FUNCTION_BLOCK FB_ActiveTarget EXTENDS FB_TargetBase IMPLEMENTS I_Device
VAR_INPUT
END_VAR
VAR_OUTPUT
END_VAR
VAR
	bInitFB			: BOOL := TRUE;
	nNotifyId		: UINT;
	bError			: BOOL;
	nErrorId		: ERRORID;
	bCanceled		: BOOL;
	bStop			: BOOL;
	bBusy			: BOOL;
	eCurrentState	: E_MachineState := E_MachineState.MACHINESTATE_Idle;
	stError			: ST_Error;
	bIsInit			: BOOL;	
	stProcessData	: ST_ObjectProcData;
	eCurrentAction	: E_Action;
	
	//Verkettete Liste für BasicActions
	fbList				: FB_LinkedListCtrl;
	hList				: T_HLINKEDLIST;
	aNodes           	: ARRAY[0..4] OF T_LinkedListEntry;
	getValue			: PVOID;
	getPosPtr       	: POINTER TO T_LinkedListEntry := 0;
	
	
	//Action: "Init"
	bInit				: BOOL;				//Action A_Init() aktiv setzen
	nStateA_Init		: USINT;			//State von A_Init()
	bFlagA_Init			: BOOL := TRUE;		//Hilfsflag A_Init()
	
	//Action: Stop
	nStateA_Stop		: USINT;	//Statemachine von A_Stop()
	bStopAllOnError		: BOOL;
	
	//Action: "Reset"
	nStateA_Reset		: USINT;	//Statemachine von A_Reset();	
END_VAR

METHOD M_CancelAction
VAR_INPUT
	eAction	: E_Action;
END_VAR
END_METHOD

METHOD M_CheckProcDataType : BOOL
VAR_INPUT
	eProcDataType : E_ProcDataType;
END_VAR
END_METHOD

METHOD M_ExeAction : ERRORID
VAR_INPUT
	refActionData	: REFERENCE TO ST_ActionData;
END_VAR
END_METHOD

METHOD M_GetActionBusy : BOOL
VAR_INPUT
	eAction	: E_Action;
END_VAR
END_METHOD

METHOD M_GetAllProps : ERRORID
VAR_INPUT
	refCmdData : REFERENCE TO ST_CmdData;
END_VAR
M_GetAllProps := SUPER^.M_GetAllProps(refCmdData);
refCmdData.aHeader[2] := nNotifyId;
END_METHOD

METHOD M_GetDevice : I_Device
VAR_INPUT
END_VAR
M_GetDevice := THIS^;
END_METHOD

METHOD M_GetProcData : DINT
VAR_INPUT
	eProcDataType : E_ProcDataType;
END_VAR
END_METHOD

METHOD M_Reset
bBusy := TRUE;
eCurrentState := E_MachineState.MACHINESTATE_Reset;
END_METHOD

METHOD M_Stop : ERRORID
//Stop braucht nur ausgeführt werden, wenn irgendwas aktiv ist
IF NOT bStop AND eCurrentState = E_MachineState.MACHINESTATE_Active THEN
	bStop := TRUE;
	fbList.A_AddHeadValue(hList := hList, putValue := E_Action.ACTION_Stop);
END_IF
END_METHOD

PROPERTY P_bBusy : BOOL
GET
P_bBusy := bBusy;
END_GET
END_PROPERTY

PROPERTY P_bCanceled : BOOL
GET
P_bCanceled := bCanceled;
END_GET
END_PROPERTY

PROPERTY P_bError : BOOL
GET
P_bError := bError;
END_GET
END_PROPERTY

PROPERTY P_bIsInit : BOOL
GET
P_bIsInit := bIsInit;
END_GET
END_PROPERTY

PROPERTY P_bStopAllOnError : BOOL
GET
P_bStopAllOnError := bStopAllOnError;
END_GET
END_PROPERTY

PROPERTY P_eCurrentState : E_MachineState
GET
P_eCurrentState := eCurrentState;
END_GET
END_PROPERTY

PROPERTY P_nErrorId : ERRORID
GET
P_nErrorID := nErrorID;
END_GET
END_PROPERTY

PROPERTY P_nNotifyId : UINT
GET
P_nNotifyId := nNotifyId;
END_GET
SET
nNotifyId := P_nNotifyId;
END_SET
END_PROPERTY

PROPERTY P_pObject : POINTER TO FB_Object
GET
P_pObject := THIS;
END_GET
END_PROPERTY

PROPERTY P_stError : ST_Error
GET
P_stError := stError;
END_GET
END_PROPERTY

END_FUNCTION_BLOCK

(* stored: Version 1.1.0.1, ProductVersion 3.1.4024.11
   POU FB_ActiveTarget: Id {f71f8edd-f391-4a79-953f-1ef5fbc17e11}, SpecialFunc None
   Method M_CancelAction: Id {259fb960-548c-47e0-a706-3237938bcacc}
   Method M_CheckProcDataType: Id {fc140985-521b-420d-b63a-4091e80d7eb5}
   Method M_ExeAction: Id {716c8509-50bf-4c86-85ed-eafa60eb7961}
   Method M_GetActionBusy: Id {9a6380bc-025b-4a37-99a3-7eb0066118f5}
   Method M_GetAllProps: Id {bd35db0b-f5db-4f94-be53-888817275f9f}
   Method M_GetDevice: Id {1acc045b-7fb2-43b1-afdb-46301bfde7fe}
   Method M_GetProcData: Id {c5fe35ab-f162-46e9-a230-5f9164983253}
   Method M_Reset: Id {53156c17-4a46-4002-b3af-bc5d6d07a4bb}
   Method M_Stop: Id {2fd9dd19-8a3e-41d4-8cae-d39f6ea2c4f5}
   Property P_bBusy: Id {76b0dc27-93e2-4f0c-8c46-1182f9e0266c}
   Get Get: Id {f0e5cbed-3bfe-4f04-9e93-28db2db1c409}
   Property P_bCanceled: Id {a2523f95-5c48-4e04-a8bc-344e88f3b58d}
   Get Get: Id {5d2c1e46-089e-4c9d-8df5-4b32e578c889}
   Property P_bError: Id {531d40a1-5514-4de8-bb35-6f7be3009006}
   Get Get: Id {b53ded85-1d01-4c62-b396-aca953357d94}
   Property P_bIsInit: Id {b921bcca-ca77-43da-8f6e-84a267199db5}
   Get Get: Id {b661a2ef-aa49-4274-aab5-6587d179fc26}
   Property P_bStopAllOnError: Id {19e7b204-f0c5-484b-8e2d-0707f459394d}
   Get Get: Id {c0e63914-7ea4-4539-966e-8649061a65a0}
   Property P_eCurrentState: Id {e959f0e8-af35-4e45-a2c9-59cebd5de9be}
   Get Get: Id {80711c4f-899f-4dca-9950-e894f3a97d09}
   Property P_nErrorId: Id {6bc192be-ee4d-491a-aaee-300ef9c989f2}
   Get Get: Id {e12f00e9-4ec0-4d30-865a-99ed3e6efbd5}
   Property P_nNotifyId: Id {5043a063-c4fe-4a50-95fe-dae7381ec7e0}
   Get Get: Id {c9a37f0d-4123-4f95-b1ae-aefb8444bb00}
   Set Set: Id {b6d7917c-f37d-4f49-89d2-a47fa6948bba}
   Property P_pObject: Id {ce810d74-28ca-4cb4-b244-55d2a6d28539}
   Get Get: Id {7144deb9-2972-4940-bd60-f94f935dbad7}
   Property P_stError: Id {56337beb-6f12-4441-ab58-c1374d7c7643}
   Get Get: Id {baac5684-bae2-4366-b394-d8d8a66af21f} *)
